TYPE errorsSt :
STRUCT
	errorName	:	STRING;
	showError	:	BOOL;
END_STRUCT
END_TYPE

(* stored: Version 1.1.0.1, ProductVersion 3.1.4024.12
   DUT errorsSt: Id {1ef6afcc-5aa4-42cc-b2c0-8f19ad6d7e1f} *)
